TYPE st_PLCtoHMI_PressureTrans :
STRUCT
    value : LREAL;
END_STRUCT
END_TYPE

(* stored: Version 1.1.0.1, ProductVersion 3.1.4024.9
   DUT st_PLCtoHMI_PressureTrans: Id {71097384-a4f9-4861-a180-2eb2ed255ceb} *)
